FUNCTION_BLOCK TeknicEIP
VAR_INPUT CONSTANT
	bEnable : BOOL;
END_VAR
VAR_OUTPUT
	pulse AT %Q* : INT; //num pulses
	
	A : BOOL; //direction (F = inwards, T = outwards)
	B : BOOL; //home bit
	clear : BOOL;
	
	brakeRelease AT %Q* : BOOL;
	
	register AT %Q* : INT;
	
	contact AT %I* : BOOL;
	
	home AT %I* : BOOL;
	outerLimit AT %I* : BOOL;
	innerLimit AT %I* : BOOL;
	done AT %I* : BOOL;	
	
	hlfb AT %I* : REAL;
	
	homeSet : BOOL;
	busy : BOOL;
	error : BOOL;
	
	position : LREAL;
	targetPos : LREAL;
END_VAR
VAR
	mode : (HOLD, TARGET, CONTINUOUS);
	
	minHoming : TON;
	
	resetTimer : TP;
	pulser : TON;
	requestedPulses : INT;
	
	step : Homing;//(IDLE, HOME_UP, HOME_FINAL, DOWN, REDO_HOME, HOME_DONE);
END_VAR
VAR_STAT CONSTANT
	resetTime : TIME := T#1000MS;
	pulseWidth : TIME := T#25MS;
	unitsPerPulse : INT := 800; //800 Teknic units per revolution
	distancePerPulse : INT := 5; //5mm per revolution
END_VAR

register.0 := bEnable;
register.1 := A;
register.2 := B;
register.3 := clear;


resetTimer(IN:= , PT:= resetTime, Q=> clear, ET=> );
IF resetTimer.IN THEN
	IF resetTimer.Q THEN
		brakeRelease := FALSE;
		pulse := 0;
	END_IF
	RETURN;
END_IF

resetTimer.IN := FALSE;

IF NOT bEnable THEN
	RETURN;
END_IF

CASE mode OF
	HOLD:
		requestedPulses := 0;
	
	TARGET:		
		IF NOT WithinTolerance(position, targetPos, distancePerPulse) THEN
			IF position < targetPos THEN
				A := TRUE;
			ELSIF position > targetPos THEN
				A := FALSE;
			END_IF
			
			requestedPulses := TO_INT(CEILING(ABS(position - targetPos)/distancePerPulse));
			
		ELSE
			requestedPulses := 0;
			mode := HOLD;
			
		END_IF
		
	CONTINUOUS:
		requestedPulses := 1;
		
END_CASE

sequence();

IF home OR innerLimit OR outerLimit THEN
	requestedPulses := 0;
	mode := HOLD;
END_IF

METHOD homingSequence : BOOL
minHoming(IN:= , PT:= T#1S, Q=> , ET=> );

IF NOT bEnable THEN
	RETURN;
END_IF

CASE step OF
	Homing.IDLE:
		pulse := 0;
		A := FALSE;
		B := FALSE;
		brakeRelease := TRUE;
		
		homeSet := FALSE;
		step := Homing.REDO;
		
	Homing.REDO: //let insertion drop to inner limit before homing
		pulse := 0;
		A := FALSE;
		B := FALSE;
		brakeRelease := TRUE;
		
		IF NOT innerLimit THEN
			step := Homing.HOME_OUT;
		END_IF
	
	Homing.HOME_OUT:
		mode := CONTINUOUS;
	
		pulse := 1;
		A := FALSE;
		B := TRUE;
		brakeRelease := TRUE;
		
		minHoming.IN := TRUE;
		
		IF NOT home AND minHoming.Q THEN
			step := Homing.DONE;
			minHoming.IN := FALSE;
		END_IF
		
	Homing.DONE:
		pulse := 0;
		A := FALSE;
		B := TRUE;
		brakeRelease := TRUE;
		
		position := 0;
		homeSet := TRUE;
		homingSequence := TRUE;
		
		mode := HOLD;
		step := Homing.IDLE;
	
END_CASE
END_METHOD

METHOD moveAbsolute : BOOL
VAR_INPUT
	targetPos : LREAL;
END_VAR
THIS^.targetPos := targetPos;
mode := TARGET;
END_METHOD

METHOD moveContinuous : BOOL
VAR_INPUT
	direction : MC_Direction;
END_VAR
IF direction = MC_Negative_Direction THEN
	A := FALSE;
ELSIF direction = MC_Positive_Direction THEN
	A := TRUE;
END_IF

mode := CONTINUOUS;
END_METHOD

METHOD reset : BOOL
VAR_INPUT
END_VAR
resetTimer.IN := TRUE;
END_METHOD

METHOD sequence : BOOL
VAR_INPUT
END_VAR
IF hlfb > -9999 THEN //is busy
	IF A THEN //positive
		position := position + (distancePerPulse * pulse);
	ELSE
		position := position - (distancePerPulse * pulse);
	END_IF
	pulse := 0;
	RETURN;
END_IF

//is free to accept new request
IF requestedPulses > 0 THEN
	pulse := requestedPulses;
END_IF
END_METHOD

METHOD stop : BOOL
VAR_INPUT
END_VAR
mode := HOLD;
END_METHOD

END_FUNCTION_BLOCK

(* stored: Version 1.1.0.1, ProductVersion 3.1.4024.11
   POU TeknicEIP: Id {82d395c8-897a-4c3b-989f-b99dc8146760}, SpecialFunc None
   Method homingSequence: Id {ed7f9015-f217-4688-b191-db86d43e2b15}
   Method moveAbsolute: Id {dc77def1-bef9-43df-afd0-8ca352bd4ae2}
   Method moveContinuous: Id {56e37924-ed1f-434c-b8b5-86f83bcd5e14}
   Method reset: Id {b78ab13d-678d-4b52-8830-ac5e90a85d68}
   Method sequence: Id {d3e76146-deb6-4a1c-bf00-057dae828590}
   Method stop: Id {b371037c-73c2-41cf-af60-cf703d5e079a} *)
